TYPE ST_TxHmi :
STRUCT
	em8000 : ST_TxHmiStewart;
	em1500 : ST_TxHmiStewart;
	mru1 : ST_TxHmiMru;
	mru2 : ST_TxHmiMru;
	comau : ST_TxHmiComau;
	winch : ST_TxHmiWinch;
	qtm : ST_TxHmiQualisys;
	phi : ARRAY [0..1] OF REAL;
	phi_t : ARRAY [0..1] OF REAL;	
	e : ARRAY [0..2] OF REAL;
	c : REAL;
END_STRUCT
END_TYPE

(* stored: Version 1.1.0.1, ProductVersion 3.1.4022.18
   DUT ST_TxHmi: Id {6be351a3-497e-469d-b641-634e507bcf6c} *)
